Staubli VAL3: Control_Lable.pgx

public program Control_Lable(string x_sMess, num& Value, num x_nTextMode)
begin
 //在屏幕中进行显示



setTextMode(0)
gotoxy(0,0)
put(x_sMess)
gotoxy(getDisplayLen(x_sMess),0)
x_nTextMode=min(max(0,x_nTextMode),3)
setTextMode(x_nTextMode)
//序号加1
put(left(toString("",Value+1)+"            ",max(8,nPanelLTopX-getDisplayLen(x_sMess)-len(toString("",Value)))))
setTextMode(0)
end
